(*

.. <legal notes>

legal notes
=================
| SPDX-FileCopyrightText: © 2025 Oleksandr Tiutyk <trofimich@gmail.com>
| SPDX-License-Identifier: LGPL-3.0-only
| For details check: LGPL-3.0-only_

.. _LGPL-3.0-only: https://www.gnu.org/licenses/lgpl-3.0.en.html

.. </legal notes>

*)

{attribute 'no_explicit_call' := 'Direct call is not allowed'} 
FUNCTION_BLOCK ABSTRACT Object IMPLEMENTS IObject

{attribute 'monitoring' := 'call'}
PROPERTY FINAL Address : PVOID
GET
Address := THIS;
END_GET
END_PROPERTY

{attribute 'monitoring' := 'call'}
PROPERTY ABSTRACT ClassName : STRING
GET
END_GET
END_PROPERTY

{attribute "object_name" := "Equals"}
METHOD Equals : BOOL
VAR_INPUT 
	object : IObject;
END_VAR
VAR
	selfPointer : POINTER TO Object;
	comparingPointer : POINTER TO Object;
END_VAR
selfPointer := THIS;

IF __QUERYPOINTER(object, comparingPointer) THEN
	Equals := selfPointer = comparingPointer;
END_IF
END_METHOD

METHOD FB_exit : BOOL
VAR_INPUT
	bInCopyCode : BOOL; // if TRUE, the exit method is called for exiting an instance that is copied afterwards (online change).
END_VAR
IF ObjectStatisticsSettings.CountObjectStatistics THEN
	ObjectStatistics.RemoveObject(THIS^);
END_IF
END_METHOD

METHOD FB_init : BOOL
VAR_INPUT
	bInitRetains : BOOL; // if TRUE, the retain variables are initialized (warm start / cold start)
	bInCopyCode : BOOL; // if TRUE, the instance afterwards gets moved into the copy code (online change)
END_VAR
IF ObjectStatisticsSettings.CountObjectStatistics THEN
	ObjectStatistics.AddObject(THIS^);
END_IF
END_METHOD

{attribute 'monitoring' := 'call'}
PROPERTY FINAL IsDynamicInstance : BOOL
GET
IsDynamicInstance := MemoryHelper.IsDynamicData(THIS, 1);
END_GET
END_PROPERTY

{attribute 'monitoring' := 'call'}
{attribute 'OPC.UA.DA.Property' := '1'}
{attribute 'OPC.UA.DA.Access' := '1'}
PROPERTY Name : WSTRING
GET
VAR
	address : PVOID;
	addressString : STRING(23);
END_VAR
address := THIS;

addressString := Tc2_Utilities.DATA_TO_HEXSTR(ADR(address), SIZEOF(address), FALSE);

StringHelper.ReplaceInSource(addressString, ' ', '');

Name := WideStringHelper.ConcatStrings255(TO_WSTRING(ClassName), " (", TO_WSTRING(addressString), ")");
END_GET
END_PROPERTY

{attribute 'monitoring' := 'call'}
PROPERTY ABSTRACT NamespaceName : STRING
GET
END_GET
END_PROPERTY

{attribute 'monitoring' := 'call'}
PROPERTY ABSTRACT Size : ULINT
GET
END_GET
END_PROPERTY

// Returns a string representation of the object for debugging and logging purposes.
// It is recommended to include key properties in a human-readable format.
METHOD ToString : WSTRING(255)
VAR_INST
	cachedResult : WSTRING(255);
END_VAR
IF cachedResult = "" THEN
	WideStringHelper.AppendToTarget255(cachedResult, TO_WSTRING(NamespaceName), ".", TO_WSTRING(ClassName));
END_IF 

ToString := cachedResult;
END_METHOD

END_FUNCTION_BLOCK

(* stored: Version 1.1.0.1
   POU Object: Id {65208310-8b3f-466c-81b7-6cce45022676}, SpecialFunc None
   Property Address: Id {fb693a32-9773-4047-aa8f-22abdeeaa290}
   Get Get: Id {9f8bbfa3-aa5e-447f-898b-426110e9c9ed}
   Property ClassName: Id {93bace28-41b5-44d6-b854-9ee3edbd382f}
   Get Get: Id {64b538df-f61f-4f5f-95f8-f82623c92e0a}
   Method Equals: Id {c147fb9a-ab41-452b-8012-567d8446205b}
   Method FB_exit: Id {2d9f8d8d-3924-4b67-aafc-98d5a0623fe6}
   Method FB_init: Id {f1b8d6f4-27df-492c-b43a-c682b4e0f7b2}
   Property IsDynamicInstance: Id {24998a7a-78a1-4ed7-9b02-1f1a03f8b719}
   Get Get: Id {13a65fb5-a1f5-4c18-8711-a901f8b8c50f}
   Property Name: Id {335dabc6-6513-4d8b-a225-099da5e07206}
   Get Get: Id {d120e015-6224-47c6-9bd9-37bee31389df}
   Property NamespaceName: Id {c3b0678c-30f0-404d-91d4-2a5aabe2e5cc}
   Get Get: Id {816ff93c-7d0c-4e8e-8788-09a43eca472a}
   Property Size: Id {e1435e8d-7dee-46fb-af88-e0c12efed32f}
   Get Get: Id {6e225585-3ad3-46c5-8df1-c249905d905a}
   Method ToString: Id {0a892b58-fb3d-4452-8b29-2d0341433629} *)
